// TIA Portal project "Queue_v000_000_001" (V16)
// 000_000_001: set up project

(* hardware
DEVICE "S7-1200 station_1"  S7-1200 Station
   slot 0: "Rack_0"  S7-1200 Rack  Rack  V1.0
   slot 1: "PLC_1"  CPU 1212C DC/DC/DC  6ES7 212-1AE40-0XB0  V4.4
*)

// ===== PLC "PLC_1"  CPU 1212C DC/DC/DC =====

VAR_GLOBAL   // PLC tag table "Default tag table"
   "Clock_Byte" AT %MB0 : Byte;
   "Clock_10Hz" AT %M0.0 : Bool;
   "Clock_5Hz" AT %M0.1 : Bool;
   "Clock_2.5Hz" AT %M0.2 : Bool;
   "Clock_2Hz" AT %M0.3 : Bool;
   "Clock_1.25Hz" AT %M0.4 : Bool;
   "Clock_1Hz" AT %M0.5 : Bool;
   "Clock_0.625Hz" AT %M0.6 : Bool;
   "Clock_0.5Hz" AT %M0.7 : Bool;
   "System_Byte" AT %MB1 : Byte;
   "FirstScan" AT %M1.0 : Bool;
   "DiagStatusUpdate" AT %M1.1 : Bool;
   "AlwaysTRUE" AT %M1.2 : Bool;
   "AlwaysFALSE" AT %M1.3 : Bool;
END_VAR

TYPE "Int[+].UDT"
   STRUCT
      add : DInt;
      data : Array[0..4] of Int;
      length : DInt;
      remove : DInt := -1;
   END_STRUCT;
END_TYPE

FUNCTION "Int[].CountOfElements" : UDInt   // FC1, SCL
{ S7_Optimized_Access := 'TRUE' }
VERSION : 0.1
   VAR_INPUT
      data : Variant;
   END_VAR
BEGIN
   #"Int[].CountOfElements" := CountOfElements(#data);
   RETURN;
END_FUNCTION

FUNCTION "DInt.RolloverIncrement" : DInt   // FC2, SCL
TITLE = Increments a Value with Rollover
{ S7_Optimized_Access := 'TRUE' }
AUTHOR : Machado
FAMILY : DInt
VERSION : 0.1
   VAR_INPUT
      value : DInt;
      rollover : DInt;
   END_VAR
BEGIN
   #"DInt.RolloverIncrement" := (#value + 1) MOD #rollover;
   RETURN;
END_FUNCTION

FUNCTION "Int[+].Clear" : String   // FC3, SCL
{ S7_Optimized_Access := 'TRUE' }
AUTHOR : Machado
FAMILY : Int[+]
VERSION : 0.1
   VAR_INPUT
      default_add_index : Int;
      default_remove_index : Int;
      null_token : Int;
   END_VAR
   VAR_IN_OUT
      buffer : "Int[+].UDT";
   END_VAR
   VAR_TEMP
      i : DInt;
      size : DInt;
   END_VAR
   VAR CONSTANT
      DONE : String := 'cleared.';
   END_VAR
BEGIN
   REGION "GET SIZE"
       #size := UDINT_TO_DINT("Int[].CountOfElements"(#buffer.data));
   END_REGION

   REGION "CLEAR DATA"
       FOR #i := 0 TO #size - 1 DO
           #buffer.data[#i] := #null_token;
       END_FOR;
   END_REGION

   REGION "CLEAR META DATA"
       #buffer.add := #default_add_index;
       #buffer.remove := #default_remove_index;
       #buffer.length := 0;
   END_REGION

   REGION "RETURN"
       #"Int[+].Clear" := #DONE;
       RETURN;
   END_REGION
END_FUNCTION

FUNCTION "Int[+].IsEmpty" : Bool   // FC4, SCL
TITLE = Int[+] Data Array Is Empty
{ S7_Optimized_Access := 'TRUE' }
AUTHOR : Machado
FAMILY : Int[+]
VERSION : 0.1
// returns true if array is empty
   VAR_INPUT
      buffer : "Int[+].UDT";
   END_VAR
BEGIN
   IF #buffer.length = 0 THEN
       #"Int[+].IsEmpty" := TRUE;
       RETURN;
   END_IF;
   #"Int[+].IsEmpty" := FALSE;
   RETURN;
END_FUNCTION

FUNCTION "Int[+].IsFull" : Bool   // FC5, SCL
TITLE = Array Is Full
{ S7_Optimized_Access := 'TRUE' }
AUTHOR : Machado
FAMILY : Int[+]
VERSION : 0.1
// returns true if array is full
   VAR_INPUT
      buffer : "Int[+].UDT";
   END_VAR
   VAR_TEMP
      size : DInt;
   END_VAR
BEGIN
   #size := UDINT_TO_DINT("Int[].CountOfElements"(#buffer.data));
   IF #buffer.length = #size THEN
       #"Int[+].IsFull" := TRUE;
       RETURN;
   END_IF;
   #"Int[+].IsFull" := FALSE;
   RETURN;
END_FUNCTION

FUNCTION "Int[+].Pop" : String   // FC6, SCL
{ S7_Optimized_Access := 'TRUE' }
AUTHOR : Machado
FAMILY : Int[+]
VERSION : 0.1
// do not use with Add
   VAR_INPUT
      null_token : Int;
   END_VAR
   VAR_OUTPUT
      value : Int;
   END_VAR
   VAR_IN_OUT
      buffer : "Int[+].UDT";
   END_VAR
   VAR CONSTANT
      ARRAY_EMPTY : String := 'array empty. no operation.';
      POPPED : String := 'popped';
   END_VAR
BEGIN
   REGION "ARRAY EMPTY"
       IF "Int[+].IsEmpty"(#buffer) THEN
           #value := #null_token;
           #"Int[+].Pop" := #ARRAY_EMPTY;
           RETURN;
       END_IF;
   END_REGION


   REGION "POP"
       #value := #buffer.data[#buffer.remove];
       #buffer.data[#buffer.remove] := #null_token;
       #buffer.add -= 1;
       #buffer.remove -= 1;
       #buffer.length -= 1;
       #"Int[+].Pop" := #POPPED;
       RETURN;
   END_REGION
END_FUNCTION

FUNCTION "Int[+].Push" : String   // FC7, SCL
{ S7_Optimized_Access := 'TRUE' }
AUTHOR : Machado
FAMILY : Int[+]
VERSION : 0.1
// dont use push with remove
   VAR_INPUT
      value : Int;
   END_VAR
   VAR_IN_OUT
      buffer : "Int[+].UDT";
   END_VAR
   VAR CONSTANT
      ARRAY_FULL : String := 'array full. no operation.';
      PUSHED : String := 'pushed.';
   END_VAR
BEGIN
   REGION "ARRAY FULL"
       IF "Int[+].IsFull"(#buffer) THEN
           #"Int[+].Push" := #ARRAY_FULL;
           RETURN;
       END_IF;
   END_REGION


   REGION "PUSH"
       #buffer.data[#buffer.add] := #value;
       #buffer.add += 1;
       #buffer.remove += 1;
       #buffer.length += 1;
       #"Int[+].Push" := #PUSHED;
       RETURN;
   END_REGION
END_FUNCTION

FUNCTION "Int[+].Remove" : String   // FC8, SCL
{ S7_Optimized_Access := 'TRUE' }
AUTHOR : Machado
FAMILY : Int[+]
VERSION : 0.1
// dont use with Int[+].Push
   VAR_INPUT
      null_token : Int;
   END_VAR
   VAR_OUTPUT
      value : Int;
   END_VAR
   VAR_IN_OUT
      buffer : "Int[+].UDT";
   END_VAR
   VAR_TEMP
      size : DInt;
   END_VAR
   VAR CONSTANT
      ARRAY_EMPTY : String := 'array  empty. no operation.';
      REMOVED : String := 'removed.';
   END_VAR
BEGIN
   REGION "ARRAY EMPTY"
       IF "Int[+].IsEmpty"(#buffer) THEN
           #value := #null_token;
           #"Int[+].Remove" := #ARRAY_EMPTY;
           RETURN;
       END_IF;
   END_REGION


   REGION "REMOVE"
       #size := UDINT_TO_DINT("Int[].CountOfElements"(#buffer.data));
       #value := #buffer.data[#buffer.remove];
       #buffer.data[#buffer.remove] := #null_token;
       #buffer.remove := "DInt.RolloverIncrement"(value := #buffer.remove,
                                                  rollover := #size);
       #buffer.length -= 1;
       #"Int[+].Remove" := #REMOVED;
       RETURN;
   END_REGION
END_FUNCTION

FUNCTION "Int[+].Add" : String   // FC9, SCL
{ S7_Optimized_Access := 'TRUE' }
AUTHOR : Machado
FAMILY : Int[+]
VERSION : 0.1
// do not use with Pop
   VAR_INPUT
      value : Int;
   END_VAR
   VAR_IN_OUT
      buffer : "Int[+].UDT";
   END_VAR
   VAR_TEMP
      size : DInt;
   END_VAR
   VAR CONSTANT
      ARRAY_FULL : String := 'array full. no operatoin.';
      ADDED : String := 'added.';
   END_VAR
BEGIN
   REGION "ARRAY FULL"
       IF "Int[+].IsFull"(#buffer) THEN
           #"Int[+].Add" := #ARRAY_FULL;
           RETURN;
       END_IF;
   END_REGION


   REGION "ADD"
       #size := UDINT_TO_DINT("Int[].CountOfElements"(#buffer.data));
       #buffer.data[#buffer.add] := #value;
       #buffer.add := "DInt.RolloverIncrement"(value := #buffer.add,
                                               rollover := #size);
       #buffer.length += 1;
       #"Int[+].Add" := #ADDED;
       RETURN;
   END_REGION
END_FUNCTION

ORGANIZATION_BLOCK "Main"   // OB1, LAD, ProgramCycle
TITLE = "Main Program Sweep (Cycle)"
{ S7_Optimized_Access := 'TRUE' }
VERSION : 0.1
   VAR_INPUT
      Initial_Call : Bool;   // Initial call of this OB
      Remanence : Bool;   // =True, if remanent data are available
   END_VAR
BEGIN
END_ORGANIZATION_BLOCK